// TIA Portal V19 export
TYPE "Positioning_MOL_Machine_Pers_Data"
// stored: Access Published
   STRUCT
      AxisHomed { S7_SetPoint := 'True'} : Bool;
   END_STRUCT;
END_TYPE
